KUKA KRL program: Draw.src, Draw.dat

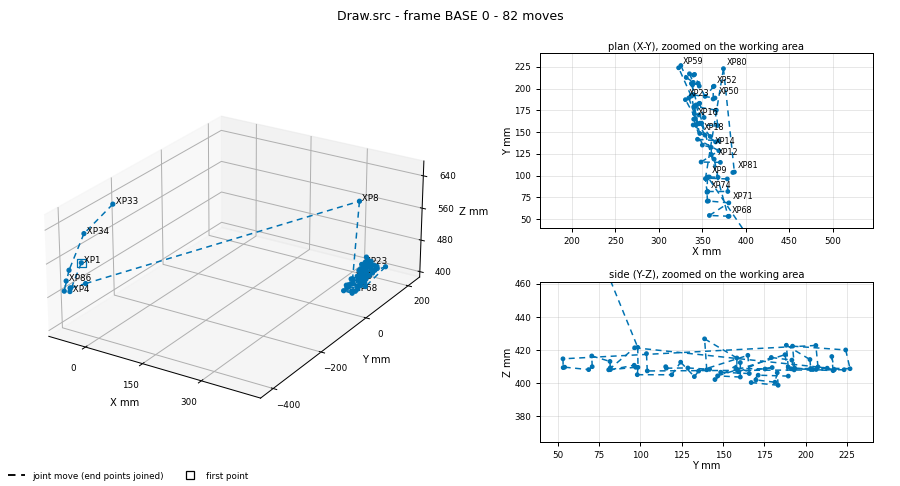
[picture p0: tool path of Draw.src in frame BASE 0, 82 of 86 moves have a stored position in this frame; points joined in program order, loops and branches not executed]
--- Draw.src ---
&ACCESS RVP
&REL 111
&PARAM EDITMASK = *
&PARAM TEMPLATE = C:\KRC\Roboter\Template\vorgabe
&PARAM DISKPATH = KRC:\R1\Program\MSROBOT
DEF BETTA( )
;FOLD INI;%{PE}
  ;FOLD BASISTECH INI
    GLOBAL INTERRUPT DECL 3 WHEN $STOPMESS==TRUE DO IR_STOPM ( )
    INTERRUPT ON 3
    BAS (#INITMOV,0 )
  ;ENDFOLD (BASISTECH INI)
  ;FOLD USER INI
    ;Make your modifications here

  ;ENDFOLD (USER INI)
;ENDFOLD (INI)

;FOLD PTP HOME  Vel= 100 % DEFAULT;%{PE}%MKUKATPBASIS,%CMOVE,%VPTP,%P 1:PTP, 2:HOME, 3:, 5:100, 7:DEFAULT
$BWDSTART = FALSE
PDAT_ACT=PDEFAULT
FDAT_ACT=FHOME
BAS (#PTP_PARAMS,100 )
$H_POS=XHOME
PTP  XHOME
;ENDFOLD

;FOLD PTP P1 Vel=100 % PDAT1 Tool[1] Base[0];%{PE}%R 8.3.48,%MKUKATPBASIS,%CMOVE,%VPTP,%P 1:PTP, 2:P1, 3:, 5:100, 7:PDAT1
$BWDSTART=FALSE
PDAT_ACT=PPDAT1
FDAT_ACT=FP1
BAS(#PTP_PARAMS,100)
PTP XP1
;ENDFOLD

;FOLD PTP P4 Vel=100 % PDAT4 Tool[1] Base[0];%{PE}%R 8.3.48,%MKUKATPBASIS,%CMOVE,%VPTP,%P 1:PTP, 2:P4, 3:, 5:100, 7:PDAT4
$BWDSTART=FALSE
PDAT_ACT=PPDAT4
FDAT_ACT=FP4
BAS(#PTP_PARAMS,100)
PTP XP4
;ENDFOLD
;FOLD Gripper SET [1]Gripper State=[2]CLOSE Wait 0.2[s] Check with Strategy 1 ;%{PE}
;FOLD Parameters Parameters ;%{h}
;Params IlfProvider=GripperTech.GripperSet;setgripper=1;setstate=2;setcont=nocont;waittime=0.2;errorstrategy=1
;ENDFOLD
GRPg_SetStateAndCheck(1, 2, 0.2, 1)
;ENDFOLD
;FOLD PTP P5 Vel=100 % PDAT5 Tool[1] Base[0];%{PE}%R 8.3.48,%MKUKATPBASIS,%CMOVE,%VPTP,%P 1:PTP, 2:P5, 3:, 5:100, 7:PDAT5
$BWDSTART=FALSE
PDAT_ACT=PPDAT5
FDAT_ACT=FP5
BAS(#PTP_PARAMS,100)
PTP XP5
;ENDFOLD
;FOLD PTP P6 Vel=100 % PDAT6 Tool[1] Base[0];%{PE}%R 8.3.48,%MKUKATPBASIS,%CMOVE,%VPTP,%P 1:PTP, 2:P6, 3:, 5:100, 7:PDAT6
$BWDSTART=FALSE
PDAT_ACT=PPDAT6
FDAT_ACT=FP6
BAS(#PTP_PARAMS,100)
PTP XP6
;ENDFOLD
;FOLD PTP P7 Vel=100 % PDAT7 Tool[1] Base[0];%{PE}%R 8.3.48,%MKUKATPBASIS,%CMOVE,%VPTP,%P 1:PTP, 2:P7, 3:, 5:100, 7:PDAT7
$BWDSTART=FALSE
PDAT_ACT=PPDAT7
FDAT_ACT=FP7
BAS(#PTP_PARAMS,100)
PTP XP7
;ENDFOLD
;FOLD PTP P8 Vel=100 % PDAT8 Tool[1] Base[0];%{PE}%R 8.3.48,%MKUKATPBASIS,%CMOVE,%VPTP,%P 1:PTP, 2:P8, 3:, 5:100, 7:PDAT8
$BWDSTART=FALSE
PDAT_ACT=PPDAT8
FDAT_ACT=FP8
BAS(#PTP_PARAMS,100)
PTP XP8
;ENDFOLD
;FOLD WAIT Time=5 sec;%{PE}%R 8.3.48,%MKUKATPBASIS,%CWAIT,%VWAIT,%P 3:5
WAIT SEC 5
;ENDFOLD
;FOLD ; print word LIFE (RAMIL AND ILIA);%{PE}%R 8.3.48,%MKUKATPBASIS,%CCOMMENT,%VNORMAL,%P 2:print word LIFE (RAMIL AND ILIA)
;ENDFOLD
;FOLD PTP P9 Vel=100 % PDAT9 Tool[1] Base[0];%{PE}%R 8.3.48,%MKUKATPBASIS,%CMOVE,%VPTP,%P 1:PTP, 2:P9, 3:, 5:100, 7:PDAT9
$BWDSTART=FALSE
PDAT_ACT=PPDAT9
FDAT_ACT=FP9
BAS(#PTP_PARAMS,100)
PTP XP9
;ENDFOLD
;FOLD PTP P10 Vel=100 % PDAT10 Tool[1] Base[0];%{PE}%R 8.3.48,%MKUKATPBASIS,%CMOVE,%VPTP,%P 1:PTP, 2:P10, 3:, 5:100, 7:PDAT10
$BWDSTART=FALSE
PDAT_ACT=PPDAT10
FDAT_ACT=FP10
BAS(#PTP_PARAMS,100)
PTP XP10
;ENDFOLD
;FOLD PTP P11 Vel=100 % PDAT11 Tool[1] Base[0];%{PE}%R 8.3.48,%MKUKATPBASIS,%CMOVE,%VPTP,%P 1:PTP, 2:P11, 3:, 5:100, 7:PDAT11
$BWDSTART=FALSE
PDAT_ACT=PPDAT11
FDAT_ACT=FP11
BAS(#PTP_PARAMS,100)
PTP XP11
;ENDFOLD
;FOLD PTP P12 Vel=100 % PDAT12 Tool[1] Base[0];%{PE}%R 8.3.48,%MKUKATPBASIS,%CMOVE,%VPTP,%P 1:PTP, 2:P12, 3:, 5:100, 7:PDAT12
$BWDSTART=FALSE
PDAT_ACT=PPDAT12
FDAT_ACT=FP12
BAS(#PTP_PARAMS,100)
PTP XP12
;ENDFOLD
;FOLD PTP P13 Vel=100 % PDAT13 Tool[1] Base[0];%{PE}%R 8.3.48,%MKUKATPBASIS,%CMOVE,%VPTP,%P 1:PTP, 2:P13, 3:, 5:100, 7:PDAT13
$BWDSTART=FALSE
PDAT_ACT=PPDAT13
FDAT_ACT=FP13
BAS(#PTP_PARAMS,100)
PTP XP13
;ENDFOLD
;FOLD PTP P14 Vel=100 % PDAT14 Tool[1] Base[0];%{PE}%R 8.3.48,%MKUKATPBASIS,%CMOVE,%VPTP,%P 1:PTP, 2:P14, 3:, 5:100, 7:PDAT14
$BWDSTART=FALSE
PDAT_ACT=PPDAT14
FDAT_ACT=FP14
BAS(#PTP_PARAMS,100)
PTP XP14
;ENDFOLD
;FOLD PTP P15 Vel=100 % PDAT15 Tool[1] Base[0];%{PE}%R 8.3.48,%MKUKATPBASIS,%CMOVE,%VPTP,%P 1:PTP, 2:P15, 3:, 5:100, 7:PDAT15
$BWDSTART=FALSE
PDAT_ACT=PPDAT15
FDAT_ACT=FP15
BAS(#PTP_PARAMS,100)
PTP XP15
;ENDFOLD
;FOLD PTP P16 Vel=100 % PDAT16 Tool[1] Base[0];%{PE}%R 8.3.48,%MKUKATPBASIS,%CMOVE,%VPTP,%P 1:PTP, 2:P16, 3:, 5:100, 7:PDAT16
$BWDSTART=FALSE
PDAT_ACT=PPDAT16
FDAT_ACT=FP16
BAS(#PTP_PARAMS,100)
PTP XP16
;ENDFOLD
;FOLD PTP P17 Vel=100 % PDAT17 Tool[1] Base[0];%{PE}%R 8.3.48,%MKUKATPBASIS,%CMOVE,%VPTP,%P 1:PTP, 2:P17, 3:, 5:100, 7:PDAT17
$BWDSTART=FALSE
PDAT_ACT=PPDAT17
FDAT_ACT=FP17
BAS(#PTP_PARAMS,100)
PTP XP17
;ENDFOLD
;FOLD PTP P18 Vel=100 % PDAT18 Tool[1] Base[0];%{PE}%R 8.3.48,%MKUKATPBASIS,%CMOVE,%VPTP,%P 1:PTP, 2:P18, 3:, 5:100, 7:PDAT18
$BWDSTART=FALSE
PDAT_ACT=PPDAT18
FDAT_ACT=FP18
BAS(#PTP_PARAMS,100)
PTP XP18
;ENDFOLD
;FOLD PTP P19 Vel=100 % PDAT19 Tool[1] Base[0];%{PE}%R 8.3.48,%MKUKATPBASIS,%CMOVE,%VPTP,%P 1:PTP, 2:P19, 3:, 5:100, 7:PDAT19
$BWDSTART=FALSE
PDAT_ACT=PPDAT19
FDAT_ACT=FP19
BAS(#PTP_PARAMS,100)
PTP XP19
;ENDFOLD
;FOLD PTP P20 Vel=100 % PDAT20 Tool[1] Base[0];%{PE}%R 8.3.48,%MKUKATPBASIS,%CMOVE,%VPTP,%P 1:PTP, 2:P20, 3:, 5:100, 7:PDAT20
$BWDSTART=FALSE
PDAT_ACT=PPDAT20
FDAT_ACT=FP20
BAS(#PTP_PARAMS,100)
PTP XP20
;ENDFOLD
;FOLD PTP P21 Vel=100 % PDAT21 Tool[1] Base[0];%{PE}%R 8.3.48,%MKUKATPBASIS,%CMOVE,%VPTP,%P 1:PTP, 2:P21, 3:, 5:100, 7:PDAT21
$BWDSTART=FALSE
PDAT_ACT=PPDAT21
FDAT_ACT=FP21
BAS(#PTP_PARAMS,100)
PTP XP21
;ENDFOLD
;FOLD PTP P22 Vel=100 % PDAT22 Tool[1] Base[0];%{PE}%R 8.3.48,%MKUKATPBASIS,%CMOVE,%VPTP,%P 1:PTP, 2:P22, 3:, 5:100, 7:PDAT22
$BWDSTART=FALSE
PDAT_ACT=PPDAT22
FDAT_ACT=FP22
BAS(#PTP_PARAMS,100)
PTP XP22
;ENDFOLD
;FOLD PTP P23 Vel=100 % PDAT23 Tool[1] Base[0];%{PE}%R 8.3.48,%MKUKATPBASIS,%CMOVE,%VPTP,%P 1:PTP, 2:P23, 3:, 5:100, 7:PDAT23
$BWDSTART=FALSE
PDAT_ACT=PPDAT23
FDAT_ACT=FP23
BAS(#PTP_PARAMS,100)
PTP XP23
;ENDFOLD
;FOLD PTP P24 Vel=100 % PDAT24 Tool[1] Base[0];%{PE}%R 8.3.48,%MKUKATPBASIS,%CMOVE,%VPTP,%P 1:PTP, 2:P24, 3:, 5:100, 7:PDAT24
$BWDSTART=FALSE
PDAT_ACT=PPDAT24
FDAT_ACT=FP24
BAS(#PTP_PARAMS,100)
PTP XP24
;ENDFOLD
;FOLD PTP P25 Vel=100 % PDAT25 Tool[1] Base[0];%{PE}%R 8.3.48,%MKUKATPBASIS,%CMOVE,%VPTP,%P 1:PTP, 2:P25, 3:, 5:100, 7:PDAT25
$BWDSTART=FALSE
PDAT_ACT=PPDAT25
FDAT_ACT=FP25
BAS(#PTP_PARAMS,100)
PTP XP25
;ENDFOLD
;FOLD PTP P26 Vel=100 % PDAT26 Tool[1] Base[0];%{PE}%R 8.3.48,%MKUKATPBASIS,%CMOVE,%VPTP,%P 1:PTP, 2:P26, 3:, 5:100, 7:PDAT26
$BWDSTART=FALSE
PDAT_ACT=PPDAT26
FDAT_ACT=FP26
BAS(#PTP_PARAMS,100)
PTP XP26
;ENDFOLD
;FOLD PTP P27 Vel=100 % PDAT27 Tool[1] Base[0];%{PE}%R 8.3.48,%MKUKATPBASIS,%CMOVE,%VPTP,%P 1:PTP, 2:P27, 3:, 5:100, 7:PDAT27
$BWDSTART=FALSE
PDAT_ACT=PPDAT27
FDAT_ACT=FP27
BAS(#PTP_PARAMS,100)
PTP XP27
;ENDFOLD
;FOLD PTP P28 Vel=100 % PDAT28 Tool[1] Base[0];%{PE}%R 8.3.48,%MKUKATPBASIS,%CMOVE,%VPTP,%P 1:PTP, 2:P28, 3:, 5:100, 7:PDAT28
$BWDSTART=FALSE
PDAT_ACT=PPDAT28
FDAT_ACT=FP28
BAS(#PTP_PARAMS,100)
PTP XP28
;ENDFOLD
;FOLD PTP P29 Vel=100 % PDAT29 Tool[1] Base[0];%{PE}%R 8.3.48,%MKUKATPBASIS,%CMOVE,%VPTP,%P 1:PTP, 2:P29, 3:, 5:100, 7:PDAT29
$BWDSTART=FALSE
PDAT_ACT=PPDAT29
FDAT_ACT=FP29
BAS(#PTP_PARAMS,100)
PTP XP29
;ENDFOLD
;FOLD PTP P30 Vel=100 % PDAT30 Tool[1] Base[0];%{PE}%R 8.3.48,%MKUKATPBASIS,%CMOVE,%VPTP,%P 1:PTP, 2:P30, 3:, 5:100, 7:PDAT30
$BWDSTART=FALSE
PDAT_ACT=PPDAT30
FDAT_ACT=FP30
BAS(#PTP_PARAMS,100)
PTP XP30
;ENDFOLD
;FOLD PTP HOME Vel=100 % DEFAULT;%{PE}%R 8.3.48,%MKUKATPBASIS,%CMOVE,%VPTP,%P 1:PTP, 2:HOME, 3:, 5:100, 7:DEFAULT
$BWDSTART=FALSE
PDAT_ACT=PDEFAULT
FDAT_ACT=FHOME
BAS(#PTP_PARAMS,100)
$H_POS=XHOME
PTP XHOME
;ENDFOLD
;FOLD ; print more (ALBERT AND ALEXANDR);%{PE}%R 8.3.48,%MKUKATPBASIS,%CCOMMENT,%VNORMAL,%P 2:print more (ALBERT AND ALEXANDR)
;ENDFOLD
;FOLD WAIT Time=2 sec;%{PE}%R 8.3.48,%MKUKATPBASIS,%CWAIT,%VWAIT,%P 3:2
WAIT SEC 2
;ENDFOLD
;FOLD PTP P36 Vel=100 % PDAT36 Tool[1] Base[0];%{PE}%R 8.3.48,%MKUKATPBASIS,%CMOVE,%VPTP,%P 1:PTP, 2:P36, 3:, 5:100, 7:PDAT36
$BWDSTART=FALSE
PDAT_ACT=PPDAT36
FDAT_ACT=FP36
BAS(#PTP_PARAMS,100)
PTP XP36
;ENDFOLD
;FOLD PTP P37 Vel=100 % PDAT37 Tool[1] Base[0];%{PE}%R 8.3.48,%MKUKATPBASIS,%CMOVE,%VPTP,%P 1:PTP, 2:P37, 3:, 5:100, 7:PDAT37
$BWDSTART=FALSE
PDAT_ACT=PPDAT37
FDAT_ACT=FP37
BAS(#PTP_PARAMS,100)
PTP XP37
;ENDFOLD
;FOLD PTP P38 Vel=100 % PDAT38 Tool[1] Base[0];%{PE}%R 8.3.48,%MKUKATPBASIS,%CMOVE,%VPTP,%P 1:PTP, 2:P38, 3:, 5:100, 7:PDAT38
$BWDSTART=FALSE
PDAT_ACT=PPDAT38
FDAT_ACT=FP38
BAS(#PTP_PARAMS,100)
PTP XP38
;ENDFOLD
;FOLD PTP P39 Vel=100 % PDAT39 Tool[1] Base[0];%{PE}%R 8.3.48,%MKUKATPBASIS,%CMOVE,%VPTP,%P 1:PTP, 2:P39, 3:, 5:100, 7:PDAT39
$BWDSTART=FALSE
PDAT_ACT=PPDAT39
FDAT_ACT=FP39
BAS(#PTP_PARAMS,100)
PTP XP39
;ENDFOLD
;FOLD PTP P40 Vel=100 % PDAT40 Tool[1] Base[0];%{PE}%R 8.3.48,%MKUKATPBASIS,%CMOVE,%VPTP,%P 1:PTP, 2:P40, 3:, 5:100, 7:PDAT40
$BWDSTART=FALSE
PDAT_ACT=PPDAT40
FDAT_ACT=FP40
BAS(#PTP_PARAMS,100)
PTP XP40
;ENDFOLD
;FOLD PTP P41 Vel=100 % PDAT41 Tool[1] Base[0];%{PE}%R 8.3.48,%MKUKATPBASIS,%CMOVE,%VPTP,%P 1:PTP, 2:P41, 3:, 5:100, 7:PDAT41
$BWDSTART=FALSE
PDAT_ACT=PPDAT41
FDAT_ACT=FP41
BAS(#PTP_PARAMS,100)
PTP XP41
;ENDFOLD
;FOLD PTP P42 Vel=100 % PDAT42 Tool[1] Base[0];%{PE}%R 8.3.48,%MKUKATPBASIS,%CMOVE,%VPTP,%P 1:PTP, 2:P42, 3:, 5:100, 7:PDAT42
$BWDSTART=FALSE
PDAT_ACT=PPDAT42
FDAT_ACT=FP42
BAS(#PTP_PARAMS,100)
PTP XP42
;ENDFOLD
;FOLD PTP P43 Vel=100 % PDAT43 Tool[1] Base[0];%{PE}%R 8.3.48,%MKUKATPBASIS,%CMOVE,%VPTP,%P 1:PTP, 2:P43, 3:, 5:100, 7:PDAT43
$BWDSTART=FALSE
PDAT_ACT=PPDAT43
FDAT_ACT=FP43
BAS(#PTP_PARAMS,100)
PTP XP43
;ENDFOLD
;FOLD PTP P44 Vel=100 % PDAT44 Tool[1] Base[0];%{PE}%R 8.3.48,%MKUKATPBASIS,%CMOVE,%VPTP,%P 1:PTP, 2:P44, 3:, 5:100, 7:PDAT44
$BWDSTART=FALSE
PDAT_ACT=PPDAT44
FDAT_ACT=FP44
BAS(#PTP_PARAMS,100)
PTP XP44
;ENDFOLD
;FOLD PTP P45 Vel=100 % PDAT45 Tool[1] Base[0];%{PE}%R 8.3.48,%MKUKATPBASIS,%CMOVE,%VPTP,%P 1:PTP, 2:P45, 3:, 5:100, 7:PDAT45
$BWDSTART=FALSE
PDAT_ACT=PPDAT45
FDAT_ACT=FP45
BAS(#PTP_PARAMS,100)
PTP XP45
;ENDFOLD
;FOLD PTP P46 Vel=100 % PDAT46 Tool[1] Base[0];%{PE}%R 8.3.48,%MKUKATPBASIS,%CMOVE,%VPTP,%P 1:PTP, 2:P46, 3:, 5:100, 7:PDAT46
$BWDSTART=FALSE
PDAT_ACT=PPDAT46
FDAT_ACT=FP46
BAS(#PTP_PARAMS,100)
PTP XP46
;ENDFOLD
;FOLD PTP P83 Vel=100 % PDAT83 Tool[1] Base[0];%{PE}%R 8.3.48,%MKUKATPBASIS,%CMOVE,%VPTP,%P 1:PTP, 2:P83, 3:, 5:100, 7:PDAT83
$BWDSTART=FALSE
PDAT_ACT=PPDAT83
FDAT_ACT=FP83
BAS(#PTP_PARAMS,100)
PTP XP83
;ENDFOLD
;FOLD PTP P47 Vel=100 % PDAT47 Tool[1] Base[0];%{PE}%R 8.3.48,%MKUKATPBASIS,%CMOVE,%VPTP,%P 1:PTP, 2:P47, 3:, 5:100, 7:PDAT47
$BWDSTART=FALSE
PDAT_ACT=PPDAT47
FDAT_ACT=FP47
BAS(#PTP_PARAMS,100)
PTP XP47
;ENDFOLD
;FOLD PTP P48 Vel=100 % PDAT48 Tool[1] Base[0];%{PE}%R 8.3.48,%MKUKATPBASIS,%CMOVE,%VPTP,%P 1:PTP, 2:P48, 3:, 5:100, 7:PDAT48
$BWDSTART=FALSE
PDAT_ACT=PPDAT48
FDAT_ACT=FP48
BAS(#PTP_PARAMS,100)
PTP XP48
;ENDFOLD
;FOLD PTP P49 Vel=100 % PDAT49 Tool[1] Base[0];%{PE}%R 8.3.48,%MKUKATPBASIS,%CMOVE,%VPTP,%P 1:PTP, 2:P49, 3:, 5:100, 7:PDAT49
$BWDSTART=FALSE
PDAT_ACT=PPDAT49
FDAT_ACT=FP49
BAS(#PTP_PARAMS,100)
PTP XP49
;ENDFOLD
;FOLD PTP P50 Vel=100 % PDAT50 Tool[1] Base[0];%{PE}%R 8.3.48,%MKUKATPBASIS,%CMOVE,%VPTP,%P 1:PTP, 2:P50, 3:, 5:100, 7:PDAT50
$BWDSTART=FALSE
PDAT_ACT=PPDAT50
FDAT_ACT=FP50
BAS(#PTP_PARAMS,100)
PTP XP50
;ENDFOLD
;FOLD PTP P51 Vel=100 % PDAT51 Tool[1] Base[0];%{PE}%R 8.3.48,%MKUKATPBASIS,%CMOVE,%VPTP,%P 1:PTP, 2:P51, 3:, 5:100, 7:PDAT51
$BWDSTART=FALSE
PDAT_ACT=PPDAT51
FDAT_ACT=FP51
BAS(#PTP_PARAMS,100)
PTP XP51
;ENDFOLD
;FOLD PTP P52 Vel=100 % PDAT52 Tool[1] Base[0];%{PE}%R 8.3.48,%MKUKATPBASIS,%CMOVE,%VPTP,%P 1:PTP, 2:P52, 3:, 5:100, 7:PDAT52
$BWDSTART=FALSE
PDAT_ACT=PPDAT52
FDAT_ACT=FP52
BAS(#PTP_PARAMS,100)
PTP XP52
;ENDFOLD
;FOLD PTP P53 Vel=100 % PDAT53 Tool[1] Base[0];%{PE}%R 8.3.48,%MKUKATPBASIS,%CMOVE,%VPTP,%P 1:PTP, 2:P53, 3:, 5:100, 7:PDAT53
$BWDSTART=FALSE
PDAT_ACT=PPDAT53
FDAT_ACT=FP53
BAS(#PTP_PARAMS,100)
PTP XP53
;ENDFOLD
;FOLD PTP P54 Vel=100 % PDAT54 Tool[1] Base[0];%{PE}%R 8.3.48,%MKUKATPBASIS,%CMOVE,%VPTP,%P 1:PTP, 2:P54, 3:, 5:100, 7:PDAT54
$BWDSTART=FALSE
PDAT_ACT=PPDAT54
FDAT_ACT=FP54
BAS(#PTP_PARAMS,100)
PTP XP54
;ENDFOLD
;FOLD PTP P55 Vel=100 % PDAT55 Tool[1] Base[0];%{PE}%R 8.3.48,%MKUKATPBASIS,%CMOVE,%VPTP,%P 1:PTP, 2:P55, 3:, 5:100, 7:PDAT55
$BWDSTART=FALSE
PDAT_ACT=PPDAT55
FDAT_ACT=FP55
BAS(#PTP_PARAMS,100)
PTP XP55
;ENDFOLD
;FOLD PTP P56 Vel=100 % PDAT56 Tool[1] Base[0];%{PE}%R 8.3.48,%MKUKATPBASIS,%CMOVE,%VPTP,%P 1:PTP, 2:P56, 3:, 5:100, 7:PDAT56
$BWDSTART=FALSE
PDAT_ACT=PPDAT56
FDAT_ACT=FP56
BAS(#PTP_PARAMS,100)
PTP XP56
;ENDFOLD
;FOLD PTP P57 Vel=100 % PDAT57 Tool[1] Base[0];%{PE}%R 8.3.48,%MKUKATPBASIS,%CMOVE,%VPTP,%P 1:PTP, 2:P57, 3:, 5:100, 7:PDAT57
$BWDSTART=FALSE
PDAT_ACT=PPDAT57
FDAT_ACT=FP57
BAS(#PTP_PARAMS,100)
PTP XP57
;ENDFOLD
;FOLD PTP P58 Vel=100 % PDAT58 Tool[1] Base[0];%{PE}%R 8.3.48,%MKUKATPBASIS,%CMOVE,%VPTP,%P 1:PTP, 2:P58, 3:, 5:100, 7:PDAT58
$BWDSTART=FALSE
PDAT_ACT=PPDAT58
FDAT_ACT=FP58
BAS(#PTP_PARAMS,100)
PTP XP58
;ENDFOLD
;FOLD PTP P59 Vel=100 % PDAT59 Tool[1] Base[0];%{PE}%R 8.3.48,%MKUKATPBASIS,%CMOVE,%VPTP,%P 1:PTP, 2:P59, 3:, 5:100, 7:PDAT59
$BWDSTART=FALSE
PDAT_ACT=PPDAT59
FDAT_ACT=FP59
BAS(#PTP_PARAMS,100)
PTP XP59
;ENDFOLD
;FOLD PTP P60 Vel=100 % PDAT60 Tool[1] Base[0];%{PE}%R 8.3.48,%MKUKATPBASIS,%CMOVE,%VPTP,%P 1:PTP, 2:P60, 3:, 5:100, 7:PDAT60
$BWDSTART=FALSE
PDAT_ACT=PPDAT60
FDAT_ACT=FP60
BAS(#PTP_PARAMS,100)
PTP XP60
;ENDFOLD
;FOLD PTP P61 Vel=100 % PDAT61 Tool[1] Base[0];%{PE}%R 8.3.48,%MKUKATPBASIS,%CMOVE,%VPTP,%P 1:PTP, 2:P61, 3:, 5:100, 7:PDAT61
$BWDSTART=FALSE
PDAT_ACT=PPDAT61
FDAT_ACT=FP61
BAS(#PTP_PARAMS,100)
PTP XP61
;ENDFOLD
;FOLD PTP P62 Vel=100 % PDAT62 Tool[1] Base[0];%{PE}%R 8.3.48,%MKUKATPBASIS,%CMOVE,%VPTP,%P 1:PTP, 2:P62, 3:, 5:100, 7:PDAT62
$BWDSTART=FALSE
PDAT_ACT=PPDAT62
FDAT_ACT=FP62
BAS(#PTP_PARAMS,100)
PTP XP62
;ENDFOLD
;FOLD PTP P63 Vel=100 % PDAT63 Tool[1] Base[0];%{PE}%R 8.3.48,%MKUKATPBASIS,%CMOVE,%VPTP,%P 1:PTP, 2:P63, 3:, 5:100, 7:PDAT63
$BWDSTART=FALSE
PDAT_ACT=PPDAT63
FDAT_ACT=FP63
BAS(#PTP_PARAMS,100)
PTP XP63
;ENDFOLD
;FOLD PTP P64 Vel=100 % PDAT64 Tool[1] Base[0];%{PE}%R 8.3.48,%MKUKATPBASIS,%CMOVE,%VPTP,%P 1:PTP, 2:P64, 3:, 5:100, 7:PDAT64
$BWDSTART=FALSE
PDAT_ACT=PPDAT64
FDAT_ACT=FP64
BAS(#PTP_PARAMS,100)
PTP XP64
;ENDFOLD
;FOLD PTP P65 Vel=100 % PDAT65 Tool[1] Base[0];%{PE}%R 8.3.48,%MKUKATPBASIS,%CMOVE,%VPTP,%P 1:PTP, 2:P65, 3:, 5:100, 7:PDAT65
$BWDSTART=FALSE
PDAT_ACT=PPDAT65
FDAT_ACT=FP65
BAS(#PTP_PARAMS,100)
PTP XP65
;ENDFOLD
;FOLD PTP P66 Vel=100 % PDAT66 Tool[1] Base[0];%{PE}%R 8.3.48,%MKUKATPBASIS,%CMOVE,%VPTP,%P 1:PTP, 2:P66, 3:, 5:100, 7:PDAT66
$BWDSTART=FALSE
PDAT_ACT=PPDAT66
FDAT_ACT=FP66
BAS(#PTP_PARAMS,100)
PTP XP66
;ENDFOLD
;FOLD PTP P67 Vel=100 % PDAT67 Tool[1] Base[0];%{PE}%R 8.3.48,%MKUKATPBASIS,%CMOVE,%VPTP,%P 1:PTP, 2:P67, 3:, 5:100, 7:PDAT67
$BWDSTART=FALSE
PDAT_ACT=PPDAT67
FDAT_ACT=FP67
BAS(#PTP_PARAMS,100)
PTP XP67
;ENDFOLD
;FOLD PTP P68 Vel=100 % PDAT68 Tool[1] Base[0];%{PE}%R 8.3.48,%MKUKATPBASIS,%CMOVE,%VPTP,%P 1:PTP, 2:P68, 3:, 5:100, 7:PDAT68
$BWDSTART=FALSE
PDAT_ACT=PPDAT68
FDAT_ACT=FP68
BAS(#PTP_PARAMS,100)
PTP XP68
;ENDFOLD
;FOLD PTP P69 Vel=100 % PDAT69 Tool[1] Base[0];%{PE}%R 8.3.48,%MKUKATPBASIS,%CMOVE,%VPTP,%P 1:PTP, 2:P69, 3:, 5:100, 7:PDAT69
$BWDSTART=FALSE
PDAT_ACT=PPDAT69
FDAT_ACT=FP69
BAS(#PTP_PARAMS,100)
PTP XP69
;ENDFOLD
;FOLD ; print word NO(Nikita);%{PE}%R 8.3.48,%MKUKATPBASIS,%CCOMMENT,%VNORMAL,%P 2:print word NO(Nikita)
;ENDFOLD
;FOLD PTP P70 Vel=100 % PDAT70 Tool[1] Base[0];%{PE}%R 8.3.48,%MKUKATPBASIS,%CMOVE,%VPTP,%P 1:PTP, 2:P70, 3:, 5:100, 7:PDAT70
$BWDSTART=FALSE
PDAT_ACT=PPDAT70
FDAT_ACT=FP70
BAS(#PTP_PARAMS,100)
PTP XP70
;ENDFOLD
;FOLD PTP P71 Vel=100 % PDAT71 Tool[1] Base[0];%{PE}%R 8.3.48,%MKUKATPBASIS,%CMOVE,%VPTP,%P 1:PTP, 2:P71, 3:, 5:100, 7:PDAT71
$BWDSTART=FALSE
PDAT_ACT=PPDAT71
FDAT_ACT=FP71
BAS(#PTP_PARAMS,100)
PTP XP71
;ENDFOLD
;FOLD PTP P72 Vel=100 % PDAT72 Tool[1] Base[0];%{PE}%R 8.3.48,%MKUKATPBASIS,%CMOVE,%VPTP,%P 1:PTP, 2:P72, 3:, 5:100, 7:PDAT72
$BWDSTART=FALSE
PDAT_ACT=PPDAT72
FDAT_ACT=FP72
BAS(#PTP_PARAMS,100)
PTP XP72
;ENDFOLD
;FOLD PTP P73 Vel=100 % PDAT73 Tool[1] Base[0];%{PE}%R 8.3.48,%MKUKATPBASIS,%CMOVE,%VPTP,%P 1:PTP, 2:P73, 3:, 5:100, 7:PDAT73
$BWDSTART=FALSE
PDAT_ACT=PPDAT73
FDAT_ACT=FP73
BAS(#PTP_PARAMS,100)
PTP XP73
;ENDFOLD
;FOLD PTP P74 Vel=100 % PDAT74 Tool[1] Base[0];%{PE}%R 8.3.48,%MKUKATPBASIS,%CMOVE,%VPTP,%P 1:PTP, 2:P74, 3:, 5:100, 7:PDAT74
$BWDSTART=FALSE
PDAT_ACT=PPDAT74
FDAT_ACT=FP74
BAS(#PTP_PARAMS,100)
PTP XP74
;ENDFOLD
;FOLD PTP P75 Vel=100 % PDAT75 Tool[1] Base[0];%{PE}%R 8.3.48,%MKUKATPBASIS,%CMOVE,%VPTP,%P 1:PTP, 2:P75, 3:, 5:100, 7:PDAT75
$BWDSTART=FALSE
PDAT_ACT=PPDAT75
FDAT_ACT=FP75
BAS(#PTP_PARAMS,100)
PTP XP75
;ENDFOLD
;FOLD PTP P76 Vel=100 % PDAT76 Tool[1] Base[0];%{PE}%R 8.3.48,%MKUKATPBASIS,%CMOVE,%VPTP,%P 1:PTP, 2:P76, 3:, 5:100, 7:PDAT76
$BWDSTART=FALSE
PDAT_ACT=PPDAT76
FDAT_ACT=FP76
BAS(#PTP_PARAMS,100)
PTP XP76
;ENDFOLD
;FOLD PTP P77 Vel=100 % PDAT77 Tool[1] Base[0];%{PE}%R 8.3.48,%MKUKATPBASIS,%CMOVE,%VPTP,%P 1:PTP, 2:P77, 3:, 5:100, 7:PDAT77
$BWDSTART=FALSE
PDAT_ACT=PPDAT77
FDAT_ACT=FP77
BAS(#PTP_PARAMS,100)
PTP XP77
;ENDFOLD
;FOLD PTP P78 Vel=100 % PDAT78 Tool[1] Base[0];%{PE}%R 8.3.48,%MKUKATPBASIS,%CMOVE,%VPTP,%P 1:PTP, 2:P78, 3:, 5:100, 7:PDAT78
$BWDSTART=FALSE
PDAT_ACT=PPDAT78
FDAT_ACT=FP78
BAS(#PTP_PARAMS,100)
PTP XP78
;ENDFOLD
;FOLD PTP P84 Vel=100 % PDAT84 Tool[1] Base[0];%{PE}%R 8.3.48,%MKUKATPBASIS,%CMOVE,%VPTP,%P 1:PTP, 2:P84, 3:, 5:100, 7:PDAT84
$BWDSTART=FALSE
PDAT_ACT=PPDAT84
FDAT_ACT=FP84
BAS(#PTP_PARAMS,100)
PTP XP84
;ENDFOLD
;FOLD PTP P79 Vel=100 % PDAT79 Tool[1] Base[0];%{PE}%R 8.3.48,%MKUKATPBASIS,%CMOVE,%VPTP,%P 1:PTP, 2:P79, 3:, 5:100, 7:PDAT79
$BWDSTART=FALSE
PDAT_ACT=PPDAT79
FDAT_ACT=FP79
BAS(#PTP_PARAMS,100)
PTP XP79
;ENDFOLD
;FOLD PTP P80 Vel=100 % PDAT80 Tool[1] Base[0];%{PE}%R 8.3.48,%MKUKATPBASIS,%CMOVE,%VPTP,%P 1:PTP, 2:P80, 3:, 5:100, 7:PDAT80
$BWDSTART=FALSE
PDAT_ACT=PPDAT80
FDAT_ACT=FP80
BAS(#PTP_PARAMS,100)
PTP XP80
;ENDFOLD
;FOLD PTP P81 Vel=100 % PDAT81 Tool[1] Base[0];%{PE}%R 8.3.48,%MKUKATPBASIS,%CMOVE,%VPTP,%P 1:PTP, 2:P81, 3:, 5:100, 7:PDAT81
$BWDSTART=FALSE
PDAT_ACT=PPDAT81
FDAT_ACT=FP81
BAS(#PTP_PARAMS,100)
PTP XP81
;ENDFOLD
;FOLD PTP P82 Vel=100 % PDAT82 Tool[1] Base[0];%{PE}%R 8.3.48,%MKUKATPBASIS,%CMOVE,%VPTP,%P 1:PTP, 2:P82, 3:, 5:100, 7:PDAT82
$BWDSTART=FALSE
PDAT_ACT=PPDAT82
FDAT_ACT=FP82
BAS(#PTP_PARAMS,100)
PTP XP82
;ENDFOLD
;FOLD PTP HOME Vel=100 % DEFAULT;%{PE}%R 8.3.48,%MKUKATPBASIS,%CMOVE,%VPTP,%P 1:PTP, 2:HOME, 3:, 5:100, 7:DEFAULT
$BWDSTART=FALSE
PDAT_ACT=PDEFAULT
FDAT_ACT=FHOME
BAS(#PTP_PARAMS,100)
$H_POS=XHOME
PTP XHOME
;ENDFOLD
;FOLD WAIT Time=3 sec;%{PE}%R 8.3.48,%MKUKATPBASIS,%CWAIT,%VWAIT,%P 3:3
WAIT SEC 3
;ENDFOLD
;FOLD PTP P33 Vel=100 % PDAT33 Tool[1] Base[0];%{PE}%R 8.3.48,%MKUKATPBASIS,%CMOVE,%VPTP,%P 1:PTP, 2:P33, 3:, 5:100, 7:PDAT33
$BWDSTART=FALSE
PDAT_ACT=PPDAT33
FDAT_ACT=FP33
BAS(#PTP_PARAMS,100)
PTP XP33
;ENDFOLD
;FOLD PTP P34 Vel=100 % PDAT34 Tool[1] Base[0];%{PE}%R 8.3.48,%MKUKATPBASIS,%CMOVE,%VPTP,%P 1:PTP, 2:P34, 3:, 5:100, 7:PDAT34
$BWDSTART=FALSE
PDAT_ACT=PPDAT34
FDAT_ACT=FP34
BAS(#PTP_PARAMS,100)
PTP XP34
;ENDFOLD
;FOLD PTP P35 Vel=100 % PDAT35 Tool[1] Base[0];%{PE}%R 8.3.48,%MKUKATPBASIS,%CMOVE,%VPTP,%P 1:PTP, 2:P35, 3:, 5:100, 7:PDAT35
$BWDSTART=FALSE
PDAT_ACT=PPDAT35
FDAT_ACT=FP35
BAS(#PTP_PARAMS,100)
PTP XP35
;ENDFOLD
;FOLD PTP P85 Vel=100 % PDAT85 Tool[1] Base[0];%{PE}%R 8.3.48,%MKUKATPBASIS,%CMOVE,%VPTP,%P 1:PTP, 2:P85, 3:, 5:100, 7:PDAT85
$BWDSTART=FALSE
PDAT_ACT=PPDAT85
FDAT_ACT=FP85
BAS(#PTP_PARAMS,100)
PTP XP85
;ENDFOLD
;FOLD Gripper SET [1]Gripper State=[1]OPEN Wait 0.2[s] Check with Strategy 1 ;%{PE}
;FOLD Parameters Parameters ;%{h}
;Params IlfProvider=GripperTech.GripperSet;setgripper=1;setstate=1;setcont=nocont;waittime=0.2;errorstrategy=1
;ENDFOLD
GRPg_SetStateAndCheck(1, 1, 0.2, 1)
;ENDFOLD
;FOLD PTP P86 Vel=100 % PDAT86 Tool[1] Base[0];%{PE}%R 8.3.48,%MKUKATPBASIS,%CMOVE,%VPTP,%P 1:PTP, 2:P86, 3:, 5:100, 7:PDAT86
$BWDSTART=FALSE
PDAT_ACT=PPDAT86
FDAT_ACT=FP86
BAS(#PTP_PARAMS,100)
PTP XP86
;ENDFOLD
;FOLD PTP HOME Vel=100 % DEFAULT;%{PE}%R 8.3.48,%MKUKATPBASIS,%CMOVE,%VPTP,%P 1:PTP, 2:HOME, 3:, 5:100, 7:DEFAULT
$BWDSTART=FALSE
PDAT_ACT=PDEFAULT
FDAT_ACT=FHOME
BAS(#PTP_PARAMS,100)
$H_POS=XHOME
PTP XHOME
;ENDFOLD
END

--- Draw.dat ---
&ACCESS RVP
&REL 111
&PARAM EDITMASK = *
&PARAM TEMPLATE = C:\KRC\Roboter\Template\vorgabe
&PARAM DISKPATH = KRC:\R1\Program\MSROBOT
DEFDAT  BETTA
;FOLD EXTERNAL DECLARATIONS;%{PE}%MKUKATPBASIS,%CEXT,%VCOMMON,%P
;FOLD BASISTECH EXT;%{PE}%MKUKATPBASIS,%CEXT,%VEXT,%P
EXT  BAS (BAS_COMMAND  :IN,REAL  :IN )
DECL INT SUCCESS
;ENDFOLD (BASISTECH EXT)
;FOLD USER EXT;%{E}%MKUKATPUSER,%CEXT,%VEXT,%P
;Make your modifications here

;ENDFOLD (USER EXT)
;ENDFOLD (EXTERNAL DECLARATIONS)
DECL BASIS_SUGG_T LAST_BASIS={POINT1[] "P86                     ",POINT2[] "P86                     ",CP_PARAMS[] "CPDAT0                  ",PTP_PARAMS[] "PDAT86                  ",CONT[] "                        ",CP_VEL[] "2.0                     ",PTP_VEL[] "100                     ",SYNC_PARAMS[] "SYNCDAT                 ",SPL_NAME[] "S0                      ",A_PARAMS[] "ADAT0                   "}
DECL E6POS XP1={X -63.5776787,Y -369.587585,Z 540.878052,A 90.6280899,B 38.1354485,C -174.883987,S 2,T 10,E1 0.0,E2 0.0,E3 0.0,E4 0.0,E5 0.0,E6 0.0}
DECL FDAT FP1={TOOL_NO 1,BASE_NO 0,IPO_FRAME #BASE,POINT2[] " ",TQ_STATE FALSE}
DECL PDAT PPDAT1={VEL 100.000,ACC 100.000,APO_DIST 100.000,GEAR_JERK 50.0000,EXAX_IGN 0}
DECL E6POS XP2={X -68.1747742,Y -395.489166,Z 482.833527,A 89.5653534,B 29.2613068,C -176.793594,S 2,T 10,E1 0.0,E2 0.0,E3 0.0,E4 0.0,E5 0.0,E6 0.0}
DECL FDAT FP2={TOOL_NO 1,BASE_NO 0,IPO_FRAME #BASE,POINT2[] " ",TQ_STATE FALSE}
DECL PDAT PPDAT2={VEL 100.000,ACC 100.000,APO_DIST 100.000,GEAR_JERK 50.0000,EXAX_IGN 0}
DECL E6POS XP3={X -50.8816795,Y -303.619751,Z 592.035156,A 90.0595474,B 27.4204693,C -177.555435,S 2,T 10,E1 0.0,E2 0.0,E3 0.0,E4 0.0,E5 0.0,E6 0.0}
DECL FDAT FP3={TOOL_NO 1,BASE_NO 0,IPO_FRAME #BASE,POINT2[] " ",TQ_STATE FALSE}
DECL PDAT PPDAT3={VEL 100.000,ACC 100.000,APO_DIST 100.000,GEAR_JERK 50.0000,EXAX_IGN 0}
DECL E6POS XP4={X -70.3313370,Y -405.710815,Z 484.144775,A 85.5909,B 25.2635117,C -179.116745,S 2,T 10,E1 0.0,E2 0.0,E3 0.0,E4 0.0,E5 0.0,E6 0.0}
DECL FDAT FP4={TOOL_NO 1,BASE_NO 0,IPO_FRAME #BASE,POINT2[] " ",TQ_STATE FALSE}
DECL PDAT PPDAT4={VEL 100.000,ACC 100.000,APO_DIST 100.000,GEAR_JERK 50.0000,EXAX_IGN 0}
DECL E6POS XP5={X -72.3102798,Y -402.118378,Z 490.503662,A 85.2627487,B 25.6180439,C -179.081940,S 2,T 10,E1 0.0,E2 0.0,E3 0.0,E4 0.0,E5 0.0,E6 0.0}
DECL FDAT FP5={TOOL_NO 1,BASE_NO 0,IPO_FRAME #BASE,POINT2[] " ",TQ_STATE FALSE}
DECL PDAT PPDAT5={VEL 100.000,ACC 100.000,APO_DIST 100.000,GEAR_JERK 50.0000,EXAX_IGN 0}
DECL E6POS XP6={X -72.8674774,Y -398.790131,Z 489.755280,A 85.0580368,B 23.2416553,C -179.360687,S 2,T 10,E1 0.0,E2 0.0,E3 0.0,E4 0.0,E5 0.0,E6 0.0}
DECL FDAT FP6={TOOL_NO 1,BASE_NO 0,IPO_FRAME #BASE,POINT2[] " ",TQ_STATE FALSE}
DECL PDAT PPDAT6={VEL 100.000,ACC 100.000,APO_DIST 100.000,GEAR_JERK 50.0000,EXAX_IGN 0}
DECL E6POS XP7={X -64.2786789,Y -355.436829,Z 485.155884,A 85.8133774,B -10.9967585,C 176.809692,S 2,T 10,E1 0.0,E2 0.0,E3 0.0,E4 0.0,E5 0.0,E6 0.0}
DECL FDAT FP7={TOOL_NO 1,BASE_NO 0,IPO_FRAME #BASE,POINT2[] " ",TQ_STATE FALSE}
DECL PDAT PPDAT7={VEL 100.000,ACC 100.000,APO_DIST 100.000,GEAR_JERK 50.0000,EXAX_IGN 0}
DECL E6POS XP8={X 423.071350,Y -0.476922095,Z 663.867371,A -0.412260592,B 74.7694778,C 0.438156366,S 6,T 27,E1 0.0,E2 0.0,E3 0.0,E4 0.0,E5 0.0,E6 0.0}
DECL FDAT FP8={TOOL_NO 1,BASE_NO 0,IPO_FRAME #BASE,POINT2[] " ",TQ_STATE FALSE}
DECL PDAT PPDAT8={VEL 100.000,ACC 100.000,APO_DIST 100.000,GEAR_JERK 50.0000,EXAX_IGN 0}
DECL E6POS XP9={X 356.112396,Y 98.4388809,Z 421.664551,A -164.061554,B 29.5813446,C 177.316650,S 2,T 11,E1 0.0,E2 0.0,E3 0.0,E4 0.0,E5 0.0,E6 0.0}
DECL FDAT FP9={TOOL_NO 1,BASE_NO 0,IPO_FRAME #BASE,POINT2[] " ",TQ_STATE FALSE}
DECL PDAT PPDAT9={VEL 100.000,ACC 100.000,APO_DIST 100.000,GEAR_JERK 50.0000,EXAX_IGN 0}
DECL E6POS XP10={X 357.860779,Y 98.5762711,Z 409.621094,A -162.948349,B 27.4036541,C 178.029694,S 2,T 11,E1 0.0,E2 0.0,E3 0.0,E4 0.0,E5 0.0,E6 0.0}
DECL FDAT FP10={TOOL_NO 1,BASE_NO 0,IPO_FRAME #BASE,POINT2[] " ",TQ_STATE FALSE}
DECL PDAT PPDAT10={VEL 100.000,ACC 100.000,APO_DIST 100.000,GEAR_JERK 50.0000,EXAX_IGN 0}
DECL E6POS XP11={X 367.941406,Y 98.1563416,Z 405.148865,A -162.500961,B 33.5004349,C 179.529129,S 2,T 11,E1 0.0,E2 0.0,E3 0.0,E4 0.0,E5 0.0,E6 0.0}
DECL FDAT FP11={TOOL_NO 1,BASE_NO 0,IPO_FRAME #BASE,POINT2[] " ",TQ_STATE FALSE}
DECL PDAT PPDAT11={VEL 100.000,ACC 100.000,APO_DIST 100.000,GEAR_JERK 50.0000,EXAX_IGN 0}
DECL E6POS XP12={X 363.463837,Y 118.981682,Z 405.119049,A -160.021790,B 34.6747246,C 179.070099,S 2,T 11,E1 0.0,E2 0.0,E3 0.0,E4 0.0,E5 0.0,E6 0.0}
DECL FDAT FP12={TOOL_NO 1,BASE_NO 0,IPO_FRAME #BASE,POINT2[] " ",TQ_STATE FALSE}
DECL PDAT PPDAT12={VEL 100.000,ACC 100.000,APO_DIST 100.000,GEAR_JERK 50.0000,EXAX_IGN 0}
DECL E6POS XP13={X 360.234467,Y 124.376480,Z 412.711609,A -159.067184,B 35.8762169,C 179.129379,S 2,T 11,E1 0.0,E2 0.0,E3 0.0,E4 0.0,E5 0.0,E6 0.0}
DECL FDAT FP13={TOOL_NO 1,BASE_NO 0,IPO_FRAME #BASE,POINT2[] " ",TQ_STATE FALSE}
DECL PDAT PPDAT13={VEL 100.000,ACC 100.000,APO_DIST 100.000,GEAR_JERK 50.0000,EXAX_IGN 0}
DECL E6POS XP14={X 360.033081,Y 132.625137,Z 404.008453,A -157.932739,B 35.2766228,C 179.157135,S 2,T 11,E1 0.0,E2 0.0,E3 0.0,E4 0.0,E5 0.0,E6 0.0}
DECL FDAT FP14={TOOL_NO 1,BASE_NO 0,IPO_FRAME #BASE,POINT2[] " ",TQ_STATE FALSE}
DECL PDAT PPDAT14={VEL 100.000,ACC 100.000,APO_DIST 100.000,GEAR_JERK 50.0000,EXAX_IGN 0}
DECL E6POS XP15={X 349.845581,Y 135.209625,Z 407.327423,A -156.753113,B 29.9789295,C 178.585098,S 2,T 11,E1 0.0,E2 0.0,E3 0.0,E4 0.0,E5 0.0,E6 0.0}
DECL FDAT FP15={TOOL_NO 1,BASE_NO 0,IPO_FRAME #BASE,POINT2[] " ",TQ_STATE FALSE}
DECL PDAT PPDAT15={VEL 100.000,ACC 100.000,APO_DIST 100.000,GEAR_JERK 50.0000,EXAX_IGN 0}
DECL E6POS XP16={X 339.956390,Y 164.945,Z 416.858398,A -152.500504,B 34.7752953,C 178.779236,S 2,T 11,E1 0.0,E2 0.0,E3 0.0,E4 0.0,E5 0.0,E6 0.0}
DECL FDAT FP16={TOOL_NO 1,BASE_NO 0,IPO_FRAME #BASE,POINT2[] " ",TQ_STATE FALSE}
DECL PDAT PPDAT16={VEL 100.000,ACC 100.000,APO_DIST 100.000,GEAR_JERK 50.0000,EXAX_IGN 0}
DECL E6POS XP17={X 341.792786,Y 165.817108,Z 405.864838,A -152.543213,B 33.0213585,C 178.702682,S 2,T 11,E1 0.0,E2 0.0,E3 0.0,E4 0.0,E5 0.0,E6 0.0}
DECL FDAT FP17={TOOL_NO 1,BASE_NO 0,IPO_FRAME #BASE,POINT2[] " ",TQ_STATE FALSE}
DECL PDAT PPDAT17={VEL 100.000,ACC 100.000,APO_DIST 100.000,GEAR_JERK 50.0000,EXAX_IGN 0}
DECL E6POS XP18={X 346.969208,Y 148.560165,Z 406.633850,A -154.966705,B 31.4723320,C 178.649765,S 2,T 11,E1 0.0,E2 0.0,E3 0.0,E4 0.0,E5 0.0,E6 0.0}
DECL FDAT FP18={TOOL_NO 1,BASE_NO 0,IPO_FRAME #BASE,POINT2[] " ",TQ_STATE FALSE}
DECL PDAT PPDAT18={VEL 100.000,ACC 100.000,APO_DIST 100.000,GEAR_JERK 50.0000,EXAX_IGN 0}
DECL E6POS XP19={X 358.972107,Y 145.068542,Z 402.220032,A -156.443802,B 37.3762131,C 179.266357,S 2,T 11,E1 0.0,E2 0.0,E3 0.0,E4 0.0,E5 0.0,E6 0.0}
DECL FDAT FP19={TOOL_NO 1,BASE_NO 0,IPO_FRAME #BASE,POINT2[] " ",TQ_STATE FALSE}
DECL PDAT PPDAT19={VEL 100.000,ACC 100.000,APO_DIST 100.000,GEAR_JERK 50.0000,EXAX_IGN 0}
DECL E6POS XP20={X 347.008118,Y 160.401550,Z 412.491486,A -153.594711,B 36.6707611,C 179.058960,S 2,T 11,E1 0.0,E2 0.0,E3 0.0,E4 0.0,E5 0.0,E6 0.0}
DECL FDAT FP20={TOOL_NO 1,BASE_NO 0,IPO_FRAME #BASE,POINT2[] " ",TQ_STATE FALSE}
DECL PDAT PPDAT20={VEL 100.000,ACC 100.000,APO_DIST 100.000,GEAR_JERK 50.0000,EXAX_IGN 0}
DECL E6POS XP21={X 349.057312,Y 160.390930,Z 403.730804,A -153.759048,B 35.5351334,C 179.028290,S 2,T 11,E1 0.0,E2 0.0,E3 0.0,E4 0.0,E5 0.0,E6 0.0}
DECL FDAT FP21={TOOL_NO 1,BASE_NO 0,IPO_FRAME #BASE,POINT2[] " ",TQ_STATE FALSE}
DECL PDAT PPDAT21={VEL 100.000,ACC 100.000,APO_DIST 100.000,GEAR_JERK 50.0000,EXAX_IGN 0}
DECL E6POS XP22={X 352.929474,Y 146.672974,Z 404.451721,A -155.859131,B 34.3024139,C 178.875565,S 2,T 11,E1 0.0,E2 0.0,E3 0.0,E4 0.0,E5 0.0,E6 0.0}
DECL FDAT FP22={TOOL_NO 1,BASE_NO 0,IPO_FRAME #BASE,POINT2[] " ",TQ_STATE FALSE}
DECL PDAT PPDAT22={VEL 100.000,ACC 100.000,APO_DIST 100.000,GEAR_JERK 50.0000,EXAX_IGN 0}
DECL E6POS XP23={X 330.405731,Y 187.418762,Z 417.246765,A -148.814148,B 36.3315773,C 178.964264,S 2,T 11,E1 0.0,E2 0.0,E3 0.0,E4 0.0,E5 0.0,E6 0.0}
DECL FDAT FP23={TOOL_NO 1,BASE_NO 0,IPO_FRAME #BASE,POINT2[] " ",TQ_STATE FALSE}
DECL PDAT PPDAT23={VEL 100.000,ACC 100.000,APO_DIST 100.000,GEAR_JERK 50.0000,EXAX_IGN 0}
DECL E6POS XP24={X 334.327271,Y 189.370438,Z 404.308228,A -148.908020,B 35.7618866,C 179.048187,S 2,T 11,E1 0.0,E2 0.0,E3 0.0,E4 0.0,E5 0.0,E6 0.0}
DECL FDAT FP24={TOOL_NO 1,BASE_NO 0,IPO_FRAME #BASE,POINT2[] " ",TQ_STATE FALSE}
DECL PDAT PPDAT24={VEL 100.000,ACC 100.000,APO_DIST 100.000,GEAR_JERK 50.0000,EXAX_IGN 0}
DECL E6POS XP25={X 340.742310,Y 171.179153,Z 404.857178,A -151.746048,B 33.7797890,C 178.810333,S 2,T 11,E1 0.0,E2 0.0,E3 0.0,E4 0.0,E5 0.0,E6 0.0}
DECL FDAT FP25={TOOL_NO 1,BASE_NO 0,IPO_FRAME #BASE,POINT2[] " ",TQ_STATE FALSE}
DECL PDAT PPDAT25={VEL 100.000,ACC 100.000,APO_DIST 100.000,GEAR_JERK 50.0000,EXAX_IGN 0}
DECL E6POS XP26={X 351.905914,Y 166.964294,Z 400.425781,A -153.180557,B 38.6468887,C 179.375061,S 2,T 11,E1 0.0,E2 0.0,E3 0.0,E4 0.0,E5 0.0,E6 0.0}
DECL FDAT FP26={TOOL_NO 1,BASE_NO 0,IPO_FRAME #BASE,POINT2[] " ",TQ_STATE FALSE}
DECL PDAT PPDAT26={VEL 100.000,ACC 100.000,APO_DIST 100.000,GEAR_JERK 50.0000,EXAX_IGN 0}
DECL E6POS XP27={X 346.822357,Y 183.238297,Z 398.758148,A -150.710281,B 40.3064499,C 179.600281,S 2,T 11,E1 0.0,E2 0.0,E3 0.0,E4 0.0,E5 0.0,E6 0.0}
DECL FDAT FP27={TOOL_NO 1,BASE_NO 0,IPO_FRAME #BASE,POINT2[] " ",TQ_STATE FALSE}
DECL PDAT PPDAT27={VEL 100.000,ACC 100.000,APO_DIST 100.000,GEAR_JERK 50.0000,EXAX_IGN 0}
DECL E6POS XP28={X 345.783173,Y 182.695969,Z 406.329102,A -150.679489,B 41.4730186,C 179.647324,S 2,T 11,E1 0.0,E2 0.0,E3 0.0,E4 0.0,E5 0.0,E6 0.0}
DECL FDAT FP28={TOOL_NO 1,BASE_NO 0,IPO_FRAME #BASE,POINT2[] " ",TQ_STATE FALSE}
DECL PDAT PPDAT28={VEL 100.000,ACC 100.000,APO_DIST 100.000,GEAR_JERK 50.0000,EXAX_IGN 0}
DECL E6POS XP29={X 342.544312,Y 181.328415,Z 400.621490,A -150.113068,B 37.2419662,C 179.670685,S 2,T 11,E1 0.0,E2 0.0,E3 0.0,E4 0.0,E5 0.0,E6 0.0}
DECL FDAT FP29={TOOL_NO 1,BASE_NO 0,IPO_FRAME #BASE,POINT2[] " ",TQ_STATE FALSE}
DECL PDAT PPDAT29={VEL 100.000,ACC 100.000,APO_DIST 100.000,GEAR_JERK 50.0000,EXAX_IGN 0}
DECL E6POS XP30={X 346.000549,Y 169.841141,Z 401.983917,A -151.865143,B 36.0128632,C 179.504333,S 2,T 11,E1 0.0,E2 0.0,E3 0.0,E4 0.0,E5 0.0,E6 0.0}
DECL FDAT FP30={TOOL_NO 1,BASE_NO 0,IPO_FRAME #BASE,POINT2[] " ",TQ_STATE FALSE}
DECL PDAT PPDAT30={VEL 100.000,ACC 100.000,APO_DIST 100.000,GEAR_JERK 50.0000,EXAX_IGN 0}
DECL E6POS XP31={X -68.5549164,Y -374.982727,Z 603.396179,A 78.5323,B 35.4639931,C 179.496185,S 2,T 34,E1 0.0,E2 0.0,E3 0.0,E4 0.0,E5 0.0,E6 0.0}
DECL FDAT FP31={TOOL_NO 1,BASE_NO 0,IPO_FRAME #BASE,POINT2[] " ",TQ_STATE FALSE}
DECL PDAT PPDAT31={VEL 100.000,ACC 100.000,APO_DIST 100.000,GEAR_JERK 50.0000,EXAX_IGN 0}
DECL E6POS XP32={X -70.0043411,Y -403.049713,Z 566.699890,A 79.1164246,B 28.9322720,C 179.644119,S 2,T 34,E1 0.0,E2 0.0,E3 0.0,E4 0.0,E5 0.0,E6 0.0}
DECL FDAT FP32={TOOL_NO 1,BASE_NO 0,IPO_FRAME #BASE,POINT2[] " ",TQ_STATE FALSE}
DECL PDAT PPDAT32={VEL 100.000,ACC 100.000,APO_DIST 100.000,GEAR_JERK 50.0000,EXAX_IGN 0}
DECL E6POS XP33={X -51.3906288,Y -262.893738,Z 644.752502,A 76.5292053,B 66.8363647,C 177.810043,S 2,T 34,E1 0.0,E2 0.0,E3 0.0,E4 0.0,E5 0.0,E6 0.0}
DECL FDAT FP33={TOOL_NO 1,BASE_NO 0,IPO_FRAME #BASE,POINT2[] " ",TQ_STATE FALSE}
DECL PDAT PPDAT33={VEL 100.000,ACC 100.000,APO_DIST 100.000,GEAR_JERK 50.0000,EXAX_IGN 0}
DECL E6POS XP34={X -61.3853912,Y -359.727020,Z 607.502563,A 79.1519928,B 38.7078781,C 179.374313,S 2,T 34,E1 0.0,E2 0.0,E3 0.0,E4 0.0,E5 0.0,E6 0.0}
DECL FDAT FP34={TOOL_NO 1,BASE_NO 0,IPO_FRAME #BASE,POINT2[] " ",TQ_STATE FALSE}
DECL PDAT PPDAT34={VEL 100.000,ACC 100.000,APO_DIST 100.000,GEAR_JERK 50.0000,EXAX_IGN 0}
DECL E6POS XP35={X -72.5088882,Y -403.481049,Z 534.060364,A 78.7907715,B 27.2317448,C 179.640228,S 2,T 34,E1 0.0,E2 0.0,E3 0.0,E4 0.0,E5 0.0,E6 0.0}
DECL FDAT FP35={TOOL_NO 1,BASE_NO 0,IPO_FRAME #BASE,POINT2[] " ",TQ_STATE FALSE}
DECL PDAT PPDAT35={VEL 100.000,ACC 100.000,APO_DIST 100.000,GEAR_JERK 50.0000,EXAX_IGN 0}
DECL E6POS XP36={X 370.606171,Y 115.318893,Z 409.989563,A -163.514145,B 19.1502228,C 179.922775,S 2,T 35,E1 0.0,E2 0.0,E3 0.0,E4 0.0,E5 0.0,E6 0.0}
DECL FDAT FP36={TOOL_NO 1,BASE_NO 0,IPO_FRAME #BASE,POINT2[] " ",TQ_STATE FALSE}
DECL PDAT PPDAT36={VEL 100.000,ACC 100.000,APO_DIST 100.000,GEAR_JERK 50.0000,EXAX_IGN 0}
DECL E6POS XP37={X 348.444580,Y 115.721970,Z 409.096558,A -162.416672,B 17.5620956,C 179.947083,S 2,T 35,E1 0.0,E2 0.0,E3 0.0,E4 0.0,E5 0.0,E6 0.0}
DECL FDAT FP37={TOOL_NO 1,BASE_NO 0,IPO_FRAME #BASE,POINT2[] " ",TQ_STATE FALSE}
DECL PDAT PPDAT37={VEL 100.000,ACC 100.000,APO_DIST 100.000,GEAR_JERK 50.0000,EXAX_IGN 0}
DECL E6POS XP38={X 368.819641,Y 128.719803,Z 409.225922,A -161.559662,B 19.2074623,C 179.921890,S 2,T 35,E1 0.0,E2 0.0,E3 0.0,E4 0.0,E5 0.0,E6 0.0}
DECL FDAT FP38={TOOL_NO 1,BASE_NO 0,IPO_FRAME #BASE,POINT2[] " ",TQ_STATE FALSE}
DECL PDAT PPDAT38={VEL 100.000,ACC 100.000,APO_DIST 100.000,GEAR_JERK 50.0000,EXAX_IGN 0}
DECL E6POS XP39={X 344.323730,Y 141.863312,Z 408.418610,A -158.398163,B 17.7827911,C 179.943741,S 2,T 35,E1 0.0,E2 0.0,E3 0.0,E4 0.0,E5 0.0,E6 0.0}
DECL FDAT FP39={TOOL_NO 1,BASE_NO 0,IPO_FRAME #BASE,POINT2[] " ",TQ_STATE FALSE}
DECL PDAT PPDAT39={VEL 100.000,ACC 100.000,APO_DIST 100.000,GEAR_JERK 50.0000,EXAX_IGN 0}
DECL E6POS XP40={X 368.507355,Y 140.114426,Z 408.113312,A -159.981796,B 19.2961330,C 179.920517,S 2,T 35,E1 0.0,E2 0.0,E3 0.0,E4 0.0,E5 0.0,E6 0.0}
DECL FDAT FP40={TOOL_NO 1,BASE_NO 0,IPO_FRAME #BASE,POINT2[] " ",TQ_STATE FALSE}
DECL PDAT PPDAT40={VEL 100.000,ACC 100.000,APO_DIST 100.000,GEAR_JERK 50.0000,EXAX_IGN 0}
DECL E6POS XP41={X 365.108551,Y 138.819580,Z 426.807098,A -159.997864,B 22.1711464,C 179.875168,S 2,T 35,E1 0.0,E2 0.0,E3 0.0,E4 0.0,E5 0.0,E6 0.0}
DECL FDAT FP41={TOOL_NO 1,BASE_NO 0,IPO_FRAME #BASE,POINT2[] " ",TQ_STATE FALSE}
DECL PDAT PPDAT41={VEL 100.000,ACC 100.000,APO_DIST 100.000,GEAR_JERK 50.0000,EXAX_IGN 0}
DECL E6POS XP42={X 339.341309,Y 158.305222,Z 415.261841,A -155.787354,B 19.1104679,C 179.923386,S 2,T 35,E1 0.0,E2 0.0,E3 0.0,E4 0.0,E5 0.0,E6 0.0}
DECL FDAT FP42={TOOL_NO 1,BASE_NO 0,IPO_FRAME #BASE,POINT2[] " ",TQ_STATE FALSE}
DECL PDAT PPDAT42={VEL 100.000,ACC 100.000,APO_DIST 100.000,GEAR_JERK 50.0000,EXAX_IGN 0}
DECL E6POS XP43={X 342.681946,Y 158.393723,Z 408.120209,A -155.984787,B 18.0765247,C 179.939255,S 2,T 35,E1 0.0,E2 0.0,E3 0.0,E4 0.0,E5 0.0,E6 0.0}
DECL FDAT FP43={TOOL_NO 1,BASE_NO 0,IPO_FRAME #BASE,POINT2[] " ",TQ_STATE FALSE}
DECL PDAT PPDAT43={VEL 100.000,ACC 100.000,APO_DIST 100.000,GEAR_JERK 50.0000,EXAX_IGN 0}
DECL E6POS XP44={X 367.323059,Y 157.694244,Z 409.071289,A -157.569092,B 19.8844318,C 179.911377,S 2,T 35,E1 0.0,E2 0.0,E3 0.0,E4 0.0,E5 0.0,E6 0.0}
DECL FDAT FP44={TOOL_NO 1,BASE_NO 0,IPO_FRAME #BASE,POINT2[] " ",TQ_STATE FALSE}
DECL PDAT PPDAT44={VEL 100.000,ACC 100.000,APO_DIST 100.000,GEAR_JERK 50.0000,EXAX_IGN 0}
DECL E6POS XP45={X 365.965240,Y 175.338165,Z 408.596741,A -155.206421,B 20.2977657,C 179.904907,S 2,T 35,E1 0.0,E2 0.0,E3 0.0,E4 0.0,E5 0.0,E6 0.0}
DECL FDAT FP45={TOOL_NO 1,BASE_NO 0,IPO_FRAME #BASE,POINT2[] " ",TQ_STATE FALSE}
DECL PDAT PPDAT45={VEL 100.000,ACC 100.000,APO_DIST 100.000,GEAR_JERK 50.0000,EXAX_IGN 0}
DECL E6POS XP46={X 340.917328,Y 179.619659,Z 409.473297,A -153.013138,B 18.8597031,C 179.927246,S 2,T 35,E1 0.0,E2 0.0,E3 0.0,E4 0.0,E5 0.0,E6 0.0}
DECL FDAT FP46={TOOL_NO 1,BASE_NO 0,IPO_FRAME #BASE,POINT2[] " ",TQ_STATE FALSE}
DECL PDAT PPDAT46={VEL 100.000,ACC 100.000,APO_DIST 100.000,GEAR_JERK 50.0000,EXAX_IGN 0}
DECL E6POS XP47={X 339.921936,Y 179.094376,Z 415.554321,A -153.018036,B 19.8147259,C 179.912460,S 2,T 35,E1 0.0,E2 0.0,E3 0.0,E4 0.0,E5 0.0,E6 0.0}
DECL FDAT FP47={TOOL_NO 1,BASE_NO 0,IPO_FRAME #BASE,POINT2[] " ",TQ_STATE FALSE}
DECL PDAT PPDAT47={VEL 100.000,ACC 100.000,APO_DIST 100.000,GEAR_JERK 50.0000,EXAX_IGN 0}
DECL E6POS XP48={X 337.291077,Y 191.537842,Z 413.951447,A -151.210709,B 19.8010464,C 179.912674,S 2,T 35,E1 0.0,E2 0.0,E3 0.0,E4 0.0,E5 0.0,E6 0.0}
DECL FDAT FP48={TOOL_NO 1,BASE_NO 0,IPO_FRAME #BASE,POINT2[] " ",TQ_STATE FALSE}
DECL PDAT PPDAT48={VEL 100.000,ACC 100.000,APO_DIST 100.000,GEAR_JERK 50.0000,EXAX_IGN 0}
DECL E6POS XP49={X 339.675446,Y 192.893951,Z 408.065338,A -151.206635,B 19.0122108,C 179.924896,S 2,T 35,E1 0.0,E2 0.0,E3 0.0,E4 0.0,E5 0.0,E6 0.0}
DECL FDAT FP49={TOOL_NO 1,BASE_NO 0,IPO_FRAME #BASE,POINT2[] " ",TQ_STATE FALSE}
DECL PDAT PPDAT49={VEL 100.000,ACC 100.000,APO_DIST 100.000,GEAR_JERK 50.0000,EXAX_IGN 0}
DECL E6POS XP50={X 364.403748,Y 189.310852,Z 409.783447,A -153.357513,B 20.8941841,C 179.895523,S 2,T 35,E1 0.0,E2 0.0,E3 0.0,E4 0.0,E5 0.0,E6 0.0}
DECL FDAT FP50={TOOL_NO 1,BASE_NO 0,IPO_FRAME #BASE,POINT2[] " ",TQ_STATE FALSE}
DECL PDAT PPDAT50={VEL 100.000,ACC 100.000,APO_DIST 100.000,GEAR_JERK 50.0000,EXAX_IGN 0}
DECL E6POS XP51={X 362.264862,Y 188.197968,Z 422.941254,A -153.369049,B 22.8296146,C 179.864532,S 2,T 35,E1 0.0,E2 0.0,E3 0.0,E4 0.0,E5 0.0,E6 0.0}
DECL FDAT FP51={TOOL_NO 1,BASE_NO 0,IPO_FRAME #BASE,POINT2[] " ",TQ_STATE FALSE}
DECL PDAT PPDAT51={VEL 100.000,ACC 100.000,APO_DIST 100.000,GEAR_JERK 50.0000,EXAX_IGN 0}
DECL E6POS XP52={X 362.525085,Y 202.446747,Z 414.317535,A -151.636139,B 22.0102634,C 179.877747,S 2,T 35,E1 0.0,E2 0.0,E3 0.0,E4 0.0,E5 0.0,E6 0.0}
DECL FDAT FP52={TOOL_NO 1,BASE_NO 0,IPO_FRAME #BASE,POINT2[] " ",TQ_STATE FALSE}
DECL PDAT PPDAT52={VEL 100.000,ACC 100.000,APO_DIST 100.000,GEAR_JERK 50.0000,EXAX_IGN 0}
DECL E6POS XP53={X 363.319855,Y 202.891220,Z 408.908539,A -151.631531,B 21.2271099,C 179.890244,S 2,T 35,E1 0.0,E2 0.0,E3 0.0,E4 0.0,E5 0.0,E6 0.0}
DECL FDAT FP53={TOOL_NO 1,BASE_NO 0,IPO_FRAME #BASE,POINT2[] " ",TQ_STATE FALSE}
DECL PDAT PPDAT53={VEL 100.000,ACC 100.000,APO_DIST 100.000,GEAR_JERK 50.0000,EXAX_IGN 0}
DECL E6POS XP54={X 352.971588,Y 191.195526,Z 408.702972,A -152.360565,B 19.9587917,C 179.910217,S 2,T 35,E1 0.0,E2 0.0,E3 0.0,E4 0.0,E5 0.0,E6 0.0}
DECL FDAT FP54={TOOL_NO 1,BASE_NO 0,IPO_FRAME #BASE,POINT2[] " ",TQ_STATE FALSE}
DECL PDAT PPDAT54={VEL 100.000,ACC 100.000,APO_DIST 100.000,GEAR_JERK 50.0000,EXAX_IGN 0}
DECL E6POS XP55={X 345.130096,Y 206.207520,Z 408.317047,A -149.946426,B 19.9450207,C 179.910431,S 2,T 35,E1 0.0,E2 0.0,E3 0.0,E4 0.0,E5 0.0,E6 0.0}
DECL FDAT FP55={TOOL_NO 1,BASE_NO 0,IPO_FRAME #BASE,POINT2[] " ",TQ_STATE FALSE}
DECL PDAT PPDAT55={VEL 100.000,ACC 100.000,APO_DIST 100.000,GEAR_JERK 50.0000,EXAX_IGN 0}
DECL E6POS XP56={X 338.571,Y 204.312531,Z 408.287750,A -149.691315,B 19.4175320,C 179.918640,S 2,T 35,E1 0.0,E2 0.0,E3 0.0,E4 0.0,E5 0.0,E6 0.0}
DECL FDAT FP56={TOOL_NO 1,BASE_NO 0,IPO_FRAME #BASE,POINT2[] " ",TQ_STATE FALSE}
DECL PDAT PPDAT56={VEL 100.000,ACC 100.000,APO_DIST 100.000,GEAR_JERK 50.0000,EXAX_IGN 0}
DECL E6POS XP57={X 339.118347,Y 193.172272,Z 409.210022,A -151.131332,B 19.1778660,C 179.922302,S 2,T 35,E1 0.0,E2 0.0,E3 0.0,E4 0.0,E5 0.0,E6 0.0}
DECL FDAT FP57={TOOL_NO 1,BASE_NO 0,IPO_FRAME #BASE,POINT2[] " ",TQ_STATE FALSE}
DECL PDAT PPDAT57={VEL 100.000,ACC 100.000,APO_DIST 100.000,GEAR_JERK 50.0000,EXAX_IGN 0}
DECL E6POS XP58={X 336.920746,Y 191.918518,Z 422.396301,A -151.142395,B 21.2248325,C 179.890259,S 2,T 35,E1 0.0,E2 0.0,E3 0.0,E4 0.0,E5 0.0,E6 0.0}
DECL FDAT FP58={TOOL_NO 1,BASE_NO 0,IPO_FRAME #BASE,POINT2[] " ",TQ_STATE FALSE}
DECL PDAT PPDAT58={VEL 100.000,ACC 100.000,APO_DIST 100.000,GEAR_JERK 50.0000,EXAX_IGN 0}
DECL E6POS XP59={X 322.606354,Y 224.035385,Z 420.104980,A -146.375610,B 24.0657692,C 179.699173,S 2,T 35,E1 0.0,E2 0.0,E3 0.0,E4 0.0,E5 0.0,E6 0.0}
DECL FDAT FP59={TOOL_NO 1,BASE_NO 0,IPO_FRAME #BASE,POINT2[] " ",TQ_STATE FALSE}
DECL PDAT PPDAT59={VEL 100.000,ACC 100.000,APO_DIST 100.000,GEAR_JERK 50.0000,EXAX_IGN 0}
DECL E6POS XP60={X 325.156189,Y 226.664383,Z 408.772858,A -146.264771,B 23.3921795,C 179.711517,S 2,T 35,E1 0.0,E2 0.0,E3 0.0,E4 0.0,E5 0.0,E6 0.0}
DECL FDAT FP60={TOOL_NO 1,BASE_NO 0,IPO_FRAME #BASE,POINT2[] " ",TQ_STATE FALSE}
DECL PDAT PPDAT60={VEL 100.000,ACC 100.000,APO_DIST 100.000,GEAR_JERK 50.0000,EXAX_IGN 0}
DECL E6POS XP61={X 331.380127,Y 212.873856,Z 409.094269,A -148.419281,B 21.6978168,C 179.753922,S 2,T 35,E1 0.0,E2 0.0,E3 0.0,E4 0.0,E5 0.0,E6 0.0}
DECL FDAT FP61={TOOL_NO 1,BASE_NO 0,IPO_FRAME #BASE,POINT2[] " ",TQ_STATE FALSE}
DECL PDAT PPDAT61={VEL 100.000,ACC 100.000,APO_DIST 100.000,GEAR_JERK 50.0000,EXAX_IGN 0}
DECL E6POS XP62={X 346.343109,Y 203.001938,Z 408.285248,A -150.793716,B 26.9061508,C 179.620682,S 2,T 35,E1 0.0,E2 0.0,E3 0.0,E4 0.0,E5 0.0,E6 0.0}
DECL FDAT FP62={TOOL_NO 1,BASE_NO 0,IPO_FRAME #BASE,POINT2[] " ",TQ_STATE FALSE}
DECL PDAT PPDAT62={VEL 100.000,ACC 100.000,APO_DIST 100.000,GEAR_JERK 50.0000,EXAX_IGN 0}
DECL E6POS XP63={X 340.918488,Y 216.441467,Z 407.592682,A -148.771729,B 28.4310093,C 179.579605,S 2,T 35,E1 0.0,E2 0.0,E3 0.0,E4 0.0,E5 0.0,E6 0.0}
DECL FDAT FP63={TOOL_NO 1,BASE_NO 0,IPO_FRAME #BASE,POINT2[] " ",TQ_STATE FALSE}
DECL PDAT PPDAT63={VEL 100.000,ACC 100.000,APO_DIST 100.000,GEAR_JERK 50.0000,EXAX_IGN 0}
DECL E6POS XP64={X 339.662079,Y 215.642914,Z 416.122528,A -148.786819,B 29.7064533,C 179.548553,S 2,T 35,E1 0.0,E2 0.0,E3 0.0,E4 0.0,E5 0.0,E6 0.0}
DECL FDAT FP64={TOOL_NO 1,BASE_NO 0,IPO_FRAME #BASE,POINT2[] " ",TQ_STATE FALSE}
DECL PDAT PPDAT64={VEL 100.000,ACC 100.000,APO_DIST 100.000,GEAR_JERK 50.0000,EXAX_IGN 0}
DECL E6POS XP65={X 335.078430,Y 217.188354,Z 408.226868,A -148.207520,B 25.3521099,C 179.661270,S 2,T 35,E1 0.0,E2 0.0,E3 0.0,E4 0.0,E5 0.0,E6 0.0}
DECL FDAT FP65={TOOL_NO 1,BASE_NO 0,IPO_FRAME #BASE,POINT2[] " ",TQ_STATE FALSE}
DECL PDAT PPDAT65={VEL 100.000,ACC 100.000,APO_DIST 100.000,GEAR_JERK 50.0000,EXAX_IGN 0}
DECL E6POS XP66={X 339.359741,Y 207.302368,Z 409.873047,A -149.733932,B 24.6254864,C 179.680634,S 2,T 35,E1 0.0,E2 0.0,E3 0.0,E4 0.0,E5 0.0,E6 0.0}
DECL FDAT FP66={TOOL_NO 1,BASE_NO 0,IPO_FRAME #BASE,POINT2[] " ",TQ_STATE FALSE}
DECL PDAT PPDAT66={VEL 100.000,ACC 100.000,APO_DIST 100.000,GEAR_JERK 50.0000,EXAX_IGN 0}
DECL E6POS XP67={X 337.265717,Y 206.021561,Z 422.824,A -149.753647,B 26.5960522,C 179.635010,S 2,T 35,E1 0.0,E2 0.0,E3 0.0,E4 0.0,E5 0.0,E6 0.0}
DECL FDAT FP67={TOOL_NO 1,BASE_NO 0,IPO_FRAME #BASE,POINT2[] " ",TQ_STATE FALSE}
DECL PDAT PPDAT67={VEL 100.000,ACC 100.000,APO_DIST 100.000,GEAR_JERK 50.0000,EXAX_IGN 0}
DECL E6POS XP68={X 379.582428,Y 53.2709579,Z 414.754059,A -173.161362,B 24.4365864,C 179.684921,S 2,T 35,E1 0.0,E2 0.0,E3 0.0,E4 0.0,E5 0.0,E6 0.0}
DECL FDAT FP68={TOOL_NO 1,BASE_NO 0,IPO_FRAME #BASE,POINT2[] " ",TQ_STATE FALSE}
DECL PDAT PPDAT68={VEL 100.000,ACC 100.000,APO_DIST 100.000,GEAR_JERK 50.0000,EXAX_IGN 0}
DECL E6POS XP69={X 380.555603,Y 53.4081268,Z 409.424744,A -173.153656,B 23.5974369,C 179.703857,S 2,T 35,E1 0.0,E2 0.0,E3 0.0,E4 0.0,E5 0.0,E6 0.0}
DECL FDAT FP69={TOOL_NO 1,BASE_NO 0,IPO_FRAME #BASE,POINT2[] " ",TQ_STATE FALSE}
DECL PDAT PPDAT69={VEL 100.000,ACC 100.000,APO_DIST 100.000,GEAR_JERK 50.0000,EXAX_IGN 0}
DECL E6POS XP70={X 357.966125,Y 54.2951355,Z 409.702332,A -172.504395,B 22.2576504,C 179.733414,S 2,T 35,E1 0.0,E2 0.0,E3 0.0,E4 0.0,E5 0.0,E6 0.0}
DECL FDAT FP70={TOOL_NO 1,BASE_NO 0,IPO_FRAME #BASE,POINT2[] " ",TQ_STATE FALSE}
DECL PDAT PPDAT70={VEL 100.000,ACC 100.000,APO_DIST 100.000,GEAR_JERK 50.0000,EXAX_IGN 0}
DECL E6POS XP71={X 380.309784,Y 68.7854156,Z 408.220459,A -170.890411,B 23.5450726,C 179.704849,S 2,T 35,E1 0.0,E2 0.0,E3 0.0,E4 0.0,E5 0.0,E6 0.0}
DECL FDAT FP71={TOOL_NO 1,BASE_NO 0,IPO_FRAME #BASE,POINT2[] " ",TQ_STATE FALSE}
DECL PDAT PPDAT71={VEL 100.000,ACC 100.000,APO_DIST 100.000,GEAR_JERK 50.0000,EXAX_IGN 0}
DECL E6POS XP72={X 356.802094,Y 70.9279404,Z 410.006226,A -169.887390,B 22.4102020,C 179.730057,S 2,T 35,E1 0.0,E2 0.0,E3 0.0,E4 0.0,E5 0.0,E6 0.0}
DECL FDAT FP72={TOOL_NO 1,BASE_NO 0,IPO_FRAME #BASE,POINT2[] " ",TQ_STATE FALSE}
DECL PDAT PPDAT72={VEL 100.000,ACC 100.000,APO_DIST 100.000,GEAR_JERK 50.0000,EXAX_IGN 0}
DECL E6POS XP73={X 355.538025,Y 70.6758347,Z 416.487061,A -169.896759,B 23.4920845,C 179.706039,S 2,T 35,E1 0.0,E2 0.0,E3 0.0,E4 0.0,E5 0.0,E6 0.0}
DECL FDAT FP73={TOOL_NO 1,BASE_NO 0,IPO_FRAME #BASE,POINT2[] " ",TQ_STATE FALSE}
DECL PDAT PPDAT73={VEL 100.000,ACC 100.000,APO_DIST 100.000,GEAR_JERK 50.0000,EXAX_IGN 0}
DECL E6POS XP74={X 355.376221,Y 81.6767197,Z 413.163727,A -168.192215,B 23.0195332,C 179.716583,S 2,T 35,E1 0.0,E2 0.0,E3 0.0,E4 0.0,E5 0.0,E6 0.0}
DECL FDAT FP74={TOOL_NO 1,BASE_NO 0,IPO_FRAME #BASE,POINT2[] " ",TQ_STATE FALSE}
DECL PDAT PPDAT74={VEL 100.000,ACC 100.000,APO_DIST 100.000,GEAR_JERK 50.0000,EXAX_IGN 0}
DECL E6POS XP75={X 356.098907,Y 81.8432922,Z 409.300507,A -168.186737,B 22.3781090,C 179.730774,S 2,T 35,E1 0.0,E2 0.0,E3 0.0,E4 0.0,E5 0.0,E6 0.0}
DECL FDAT FP75={TOOL_NO 1,BASE_NO 0,IPO_FRAME #BASE,POINT2[] " ",TQ_STATE FALSE}
DECL PDAT PPDAT75={VEL 100.000,ACC 100.000,APO_DIST 100.000,GEAR_JERK 50.0000,EXAX_IGN 0}
DECL E6POS XP76={X 379.135681,Y 81.8583374,Z 408.195374,A -168.959869,B 23.6381454,C 179.702774,S 2,T 35,E1 0.0,E2 0.0,E3 0.0,E4 0.0,E5 0.0,E6 0.0}
DECL FDAT FP76={TOOL_NO 1,BASE_NO 0,IPO_FRAME #BASE,POINT2[] " ",TQ_STATE FALSE}
DECL PDAT PPDAT76={VEL 100.000,ACC 100.000,APO_DIST 100.000,GEAR_JERK 50.0000,EXAX_IGN 0}
DECL E6POS XP77={X 378.564056,Y 96.2830048,Z 410.860229,A -166.879639,B 24.2776546,C 179.688354,S 2,T 35,E1 0.0,E2 0.0,E3 0.0,E4 0.0,E5 0.0,E6 0.0}
DECL FDAT FP77={TOOL_NO 1,BASE_NO 0,IPO_FRAME #BASE,POINT2[] " ",TQ_STATE FALSE}
DECL PDAT PPDAT77={VEL 100.000,ACC 100.000,APO_DIST 100.000,GEAR_JERK 50.0000,EXAX_IGN 0}
DECL E6POS XP78={X 355.695770,Y 97.2106705,Z 409.630646,A -165.847412,B 22.6357803,C 179.725082,S 2,T 35,E1 0.0,E2 0.0,E3 0.0,E4 0.0,E5 0.0,E6 0.0}
DECL FDAT FP78={TOOL_NO 1,BASE_NO 0,IPO_FRAME #BASE,POINT2[] " ",TQ_STATE FALSE}
DECL PDAT PPDAT78={VEL 100.000,ACC 100.000,APO_DIST 100.000,GEAR_JERK 50.0000,EXAX_IGN 0}
DECL E6POS XP79={X 353.385620,Y 96.5777664,Z 421.433319,A -165.864883,B 24.5809689,C 179.681458,S 2,T 35,E1 0.0,E2 0.0,E3 0.0,E4 0.0,E5 0.0,E6 0.0}
DECL FDAT FP79={TOOL_NO 1,BASE_NO 0,IPO_FRAME #BASE,POINT2[] " ",TQ_STATE FALSE}
DECL PDAT PPDAT79={VEL 100.000,ACC 100.000,APO_DIST 100.000,GEAR_JERK 50.0000,EXAX_IGN 0}
DECL E6POS XP80={X 374.131592,Y 223.073822,Z 408.148346,A -150.380966,B 27.5431,C 179.612335,S 2,T 35,E1 0.0,E2 0.0,E3 0.0,E4 0.0,E5 0.0,E6 0.0}
DECL FDAT FP80={TOOL_NO 1,BASE_NO 0,IPO_FRAME #BASE,POINT2[] " ",TQ_STATE FALSE}
DECL PDAT PPDAT80={VEL 100.000,ACC 100.000,APO_DIST 100.000,GEAR_JERK 50.0000,EXAX_IGN 0}
DECL E6POS XP81={X 386.687683,Y 104.196678,Z 407.423737,A -166.071152,B 24.4366951,C 179.684738,S 2,T 35,E1 0.0,E2 0.0,E3 0.0,E4 0.0,E5 0.0,E6 0.0}
DECL FDAT FP81={TOOL_NO 1,BASE_NO 0,IPO_FRAME #BASE,POINT2[] " ",TQ_STATE FALSE}
DECL PDAT PPDAT81={VEL 100.000,ACC 100.000,APO_DIST 100.000,GEAR_JERK 50.0000,EXAX_IGN 0}
DECL E6POS XP82={X 384.886261,Y 103.710167,Z 417.891479,A -166.086639,B 26.0164413,C 179.648392,S 2,T 35,E1 0.0,E2 0.0,E3 0.0,E4 0.0,E5 0.0,E6 0.0}
DECL FDAT FP82={TOOL_NO 1,BASE_NO 0,IPO_FRAME #BASE,POINT2[] " ",TQ_STATE FALSE}
DECL PDAT PPDAT82={VEL 100.000,ACC 100.000,APO_DIST 100.000,GEAR_JERK 50.0000,EXAX_IGN 0}
DECL E6POS XP83={X 344.317139,Y 159.453110,Z 406.917572,A -155.943039,B 18.0039539,C 179.940353,S 2,T 35,E1 0.0,E2 0.0,E3 0.0,E4 0.0,E5 0.0,E6 0.0}
DECL FDAT FP83={TOOL_NO 1,BASE_NO 0,IPO_FRAME #BASE,POINT2[] " ",TQ_STATE FALSE}
DECL PDAT PPDAT83={VEL 100.000,ACC 100.000,APO_DIST 100.000,GEAR_JERK 50.0000,EXAX_IGN 0}
DECL E6POS XP84={X 355.353333,Y 80.9007645,Z 408.108368,A -168.302597,B 22.1122417,C 179.736603,S 2,T 35,E1 0.0,E2 0.0,E3 0.0,E4 0.0,E5 0.0,E6 0.0}
DECL FDAT FP84={TOOL_NO 1,BASE_NO 0,IPO_FRAME #BASE,POINT2[] " ",TQ_STATE FALSE}
DECL PDAT PPDAT84={VEL 100.000,ACC 100.000,APO_DIST 100.000,GEAR_JERK 50.0000,EXAX_IGN 0}
DECL E6POS XP85={X -74.9183884,Y -420.108551,Z 489.768097,A 78.6088257,B 19.7081642,C 179.274109,S 2,T 42,E1 0.0,E2 0.0,E3 0.0,E4 0.0,E5 0.0,E6 0.0}
DECL FDAT FP85={TOOL_NO 1,BASE_NO 0,IPO_FRAME #BASE,POINT2[] " ",TQ_STATE FALSE}
DECL PDAT PPDAT85={VEL 100.000,ACC 100.000,APO_DIST 100.000,GEAR_JERK 50.0000,EXAX_IGN 0}
DECL E6POS XP86={X -75.3587189,Y -411.292328,Z 510.622437,A 78.3040543,B 23.3165665,C 179.195969,S 2,T 42,E1 0.0,E2 0.0,E3 0.0,E4 0.0,E5 0.0,E6 0.0}
DECL FDAT FP86={TOOL_NO 1,BASE_NO 0,IPO_FRAME #BASE,POINT2[] " ",TQ_STATE FALSE}
DECL PDAT PPDAT86={VEL 100.000,ACC 100.000,APO_DIST 100.000,GEAR_JERK 50.0000,EXAX_IGN 0}
ENDDAT
